FUNCTION_BLOCK FB_MoveStepperRel
VAR_INPUT
	stepsToMove				: INT;
	PosCurrent				: UDINT;
END_VAR
VAR_OUTPUT
END_VAR
VAR
	Step 					: INT := 0;
	bPowerOn				: INT;
END_VAR

MAIN.fbAxis1.bEnable := TRUE;

CASE Step OF
0:
	//MAIN.fbAxis1.moveRelDist := 0.0;
	//MAIN.fbAxis1.moveRelVel := 0.0;
	//MAIN.fbAxis1.bMoveRelExe := FALSE;
	MAIN.fbAxis1.bHaltExe := FALSE;
	Step := 1;
1:

	IF MAIN.fbAxis1.bPwrStatus THEN
		MAIN.fbAxis1.moveRelDist := stepsToMove;
		MAIN.fbAxis1.moveRelVel := 100;
		MAIN.fbAxis1.bMoveRelExe := TRUE;
		IF MAIN.fbAxis1.bMoveRelDone THEN
			MAIN.fbAxis1.bMoveRelExe := FALSE;
			MAIN.fbAxis1.bHaltExe := TRUE;
			Step := 2;
		END_IF
	END_IF	
2:
	IF MAIN.fbAxis1.bHaltDone = TRUE THEN
		MAIN.fbAxis1.bHaltExe := FALSE;
	END_IF

	MAIN.bMoveRelative := FALSE;
	
	Step := 0;
END_CASE

END_FUNCTION_BLOCK

(* stored: Version 1.1.0.1, ProductVersion 3.1.4024.9
   POU FB_MoveStepperRel: Id {0bea6b41-c696-4199-8c4b-86405a4a07f9}, SpecialFunc None *)
